FUNCTION_BLOCK uart (* uart for RPI /dev/ttyAMA0 Parity Check: None DB: 8 stop bit 1 *)
  (* Standard: 61499-2 *)
  (* Version 0.0, 2018-03-23, 4DIAC-IDE, 4DIAC-Consortium *)
  (* Version 1.0, 2016-05-26, AZ, fortiss GmbH *)
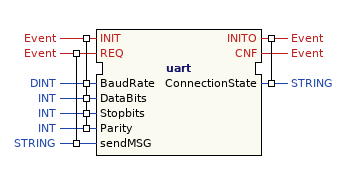
  EVENT_INPUT
    INIT WITH BaudRate, DataBits, Stopbits, Parity; (* Initialization Request *)
    REQ WITH sendMSG; (* Normal Execution Request *)
  END_EVENT
  EVENT_OUTPUT
    INITO WITH ConnectionState; (* Initialization Confirm *)
    CNF; (* Execution Confirmation *)
  END_EVENT
  VAR_INPUT
    BaudRate : DINT := 115200;
    DataBits : INT := 8; (* 7 or 8 generally select 8 *)
    Stopbits : INT := 1; (* 1 or 2 generally select 1 *)
    Parity : INT := 1; (* 1-N, 2-E, 3-O,4-S,generally select 1 *)
    sendMSG : STRING;
  END_VAR
  VAR_OUTPUT
    ConnectionState : STRING;
  END_VAR
  VAR
    fd : INT; (* Internal Variable *)
  END_VAR
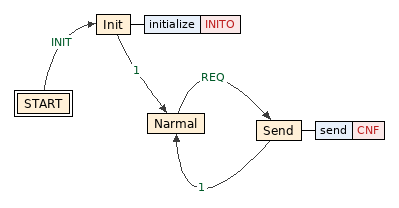
  EC_STATES
    START; (* Initial State *)
    Init : initialize -> INITO; (* Initialization *)
    Send : send -> CNF;
    Narmal;
  END_STATES
  EC_TRANSITIONS
    START TO Init := INIT;
    Narmal TO Send := REQ;
    Send TO Narmal := 1;
    Init TO Narmal := 1;
  END_TRANSITIONS
  ALGORITHM initialize IN ST: (* Initialization algorithm *)
BaudRate:=fd;
ConnectionState:="OK";
  END_ALGORITHM
  ALGORITHM send IN ST: (* Normally executed algorithm *)
sendMSG:="hello";

sendMSG:= '';
  END_ALGORITHM
END_FUNCTION_BLOCK
